TYPE ST_Recipe :
	STRUCT
		PullWheels : ST_PullWheelsRecipe;
		Sealer	   : ST_SealerRecipe;
		Unwind	   : ST_UnwindRecipe;
	END_STRUCT
END_TYPE

(* stored: Version 1.1.0.1, ProductVersion 3.1.4026.18
   DUT ST_Recipe: Id {9dbe901c-4665-4bd5-96ed-f1f6547641b0} *)
